PROGRAM PRG_TXI_VAC
VAR
END_VAR

// MSK275 Gauges
fb_ST1L1_GPI_01(PG=>st_ST1L1_GPI_01);

// MSK 500 Gauges
fb_ST1L1_GCC_01(PG := fb_ST1L1_GPI_01.PG, bEP := TRUE, IG=>st_ST1L1_GCC_01);

END_PROGRAM

(* stored: Version 1.1.0.1, ProductVersion 3.1.4024.6
   POU PRG_TXI_VAC: Id {80e6a8be-3822-46f9-baac-97367240f381}, SpecialFunc None *)
